// TIA Portal V17 export
// export: Created 2022-07-20T06:59:43.6943955Z, ExportSetting WithDefaults, DisplayName Totally Integrated Automation Portal, DisplayVersion V17, DisplayName TIA Portal Openness, DisplayVersion V17, DisplayName TIA Portal Version Control Interface, DisplayVersion V17, DisplayName SINAMICS Startdrive Advanced, DisplayVersion V17, DisplayName SINAMICS Startdrive G130, G150, S120, S150, SINAMICS MV, S210, DisplayVersion V17, DisplayName SINAMICS Startdrive G110M, G120, G120C, G120D, G120P, G115D, DisplayVersion V17, DisplayName STEP 7 Professional, DisplayVersion V17, DisplayName STEP 7 Safety, DisplayVersion V17, DisplayName WinCC Advanced, DisplayVersion V17
FUNCTION_BLOCK "FB10075_AirExtractorManager"   // FB10075, LAD
TITLE = FB10075_AirExtractorManager
{ S7_Optimized_Access := 'TRUE' }
AUTHOR : Jonathan
FAMILY : 1007x_DRYER_UV
VERSION : 1.1
// Release note: 
// 1.0 -  Alpajet version. Only analog output value
// 1.1 -  Iris improvment. Add PWM freq control
// stored: AutoNumber false, IsIECCheckEnabled false, IsRetainMemResEnabled false, MemoryReserve 100, SetENOAutomatically false, UDAEnableTagReadback false
   VAR_INPUT
      UVReady : Bool;
      UVFeedbackPower : Real;
      UVEnabled : Bool;
      AirExtractionActivation : Bool;
      ForceAirAfterShutdownUV : Bool;
      ShutterOpen : Bool;
      ShutterClose : Bool;
      ScalingShutterOpen : "stAirExtractorScalingParameters";
      ScalingShutterClosed : "stAirExtractorScalingParameters";
      PwmMinFrequenceValue : Real;
      PwmMaxFrequenceValue : Real;
   END_VAR
   VAR_OUTPUT
      AirExtractionEnable : Bool;
      AirExractionAnalogPowerValue : Int;
      ForcingAirInProgress : Bool;
      PWM_Channel_SW_Enable : Bool;
      PWM_ProgressAccel : Bool;
      PWM_FrequencyValue : Real;
   END_VAR
   VAR
      CoolingAfterClosing : Bool;
      RTrig_ShutterClose { S7_SetPoint := 'True'} : R_TRIG;
      RTrig_ForceAir { S7_SetPoint := 'True'} : R_TRIG;
      TOF_ForceAirTimer { S7_SetPoint := 'True'} : TOF_TIME;
      MemUVEnabledOnce : Bool;
      LocalPercentageValue : Real;
   END_VAR
BEGIN

REGION Network 1 (SCL): Scale Dryer Uv Power Calculation
   // Rising edge shutter closed
   #RTrig_ShutterClose(CLK := #ShutterClose);
   // Force cooling until UV Ready
   IF #RTrig_ShutterClose.Q THEN
       #CoolingAfterClosing := TRUE;
   END_IF;

   // Reset cooling if UV Ready
   IF (#UVFeedbackPower/276.48) <= #ScalingShutterClosed.PowerXMin OR #ScalingShutterClosed.PowerXMin = 0.0 THEN
       #CoolingAfterClosing := FALSE;
   END_IF;

   // Memorisation if UV was enabled one time at least
   IF #UVEnabled THEN
       #MemUVEnabledOnce := TRUE;
   END_IF;

   IF #TOF_ForceAirTimer.Q THEN
       #MemUVEnabledOnce := FALSE;
       #ForcingAirInProgress := TRUE;
   ELSE
       #ForcingAirInProgress := FALSE;
   END_IF;

   // Rising edge on force Air
   #RTrig_ForceAir(CLK := #ForceAirAfterShutdownUV);
   #TOF_ForceAirTimer(IN := #RTrig_ForceAir.Q AND #MemUVEnabledOnce,
                      PT := T#5m);

   // Air Extraction enable
   IF (#AirExtractionActivation AND #UVReady) OR #TOF_ForceAirTimer.Q THEN
       #AirExtractionEnable := TRUE;
   ELSE
       #AirExtractionEnable := FALSE;
   END_IF;


   // Scaling 
   IF #CoolingAfterClosing OR #TOF_ForceAirTimer.Q THEN
       // Force cooling after closing until UV Ready or After shutdown UV

       // Analog output
       #AirExractionAnalogPowerValue := 27648;

       // PWM Output
       #PWM_Channel_SW_Enable := TRUE;
       #PWM_FrequencyValue := #PwmMaxFrequenceValue;

   ELSIF #ShutterClose AND #AirExtractionEnable THEN
       "FC10070_ScalingAirExtraction"(SetPoint := (#UVFeedbackPower / 276.48),
                                     X_UVPower_Min := #ScalingShutterClosed.PowerXMin,
                                     X_UVPower_Max := #ScalingShutterClosed.PowerXMax,
                                     Y_AirPower_Min := #ScalingShutterClosed.PowerAirYMin,
                                     Y_AirPower_Max := #ScalingShutterClosed.PowerAirYMax,
                                     PWM_Minimum:=2000.0,
                                     PWM_Maximum:=6000.0,
                                     AnalogValue => #AirExractionAnalogPowerValue,
                                     PwmFrequenceValue => #PWM_FrequencyValue);
       #PWM_Channel_SW_Enable := TRUE;

   ELSIF #ShutterOpen AND #AirExtractionEnable THEN
       "FC10070_ScalingAirExtraction"(SetPoint := (#UVFeedbackPower / 276.48),
                                     X_UVPower_Min := #ScalingShutterOpen.PowerXMin,
                                     X_UVPower_Max := #ScalingShutterOpen.PowerXMax,
                                     Y_AirPower_Min := #ScalingShutterOpen.PowerAirYMin,
                                     Y_AirPower_Max := #ScalingShutterOpen.PowerAirYMax,
                                     PWM_Minimum:=2000.0,
                                     PWM_Maximum:=6000.0,
                                     AnalogValue => #AirExractionAnalogPowerValue,
                                     PwmFrequenceValue => #PWM_FrequencyValue);
       #PWM_Channel_SW_Enable := TRUE;
   ELSE
       #AirExractionAnalogPowerValue := 0;

       #PWM_Channel_SW_Enable := FALSE;
       #PWM_FrequencyValue := 0.0;

   END_IF;
END_REGION
END_FUNCTION_BLOCK
